// TIA Portal V17 export
// export: Created 2023-04-11T09:33:32.0254359Z, ExportSetting WithDefaults, DisplayName Totally Integrated Automation Portal, DisplayVersion V17 Update 3, DisplayName TIA Portal Openness, DisplayVersion V17 Update 3, DisplayName TIA Portal Version Control Interface, DisplayVersion V17, DisplayName SINAMICS Startdrive Advanced, DisplayVersion V17 Update2, DisplayName SINAMICS Startdrive G130, G150, S120, S150, SINAMICS MV, S210, DisplayVersion V17 Update2, DisplayName SINAMICS Startdrive G110M, G120, G120C, G120D, G120P, G115D, DisplayVersion V17 Update2, DisplayName STEP 7 Professional, DisplayVersion V17 Update 3, DisplayName STEP 7 Safety, DisplayVersion V17, DisplayName WinCC UA Professional, DisplayVersion V17 Update 3
FUNCTION "FC_and4" : Void   // FC27, FBD
{ S7_Optimized_Access := 'TRUE' }
VERSION : 0.1
// stored: AutoNumber true, IsIECCheckEnabled false, SetENOAutomatically false, UDAEnableTagReadback false
   VAR_INPUT
      in1 : Bool;
      in2 : Bool;
      in3 : Bool;
      in4 : Bool;
   END_VAR
   VAR_OUTPUT
      out : Bool;
   END_VAR
BEGIN

REGION Network 1
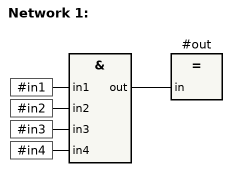
   #out := #in1 AND #in2 AND #in3 AND #in4;
END_REGION
END_FUNCTION
